# EPICS IOC start-up script: iocsh/ethercatmcAnalogOutputGenericV1.iocsh
ethercatmcCreateAsynParam $(MOTOR_PORT) $(ASYNPARAMNAME)      Float64

dbLoadRecords("ethercatmcAnalogOutputGeneric.template", "P=$(P), R=$(R), MOTOR_PORT=$(MOTOR_PORT), CHNO=$(CHNO), ASYNPARAMNAME=$(ASYNPARAMNAME), PREC=$(PREC), DESC=$(DESC), EGU=$(EGU), ASLO=$(ASLO), AOFF=$(AOFF), READBACK=$(READBACK), INITIAL_READBACK="$(INITIAL_READBACK))
